INTERFACE ITest

METHOD TestMethod : BOOL
VAR_INPUT
END_VAR
END_METHOD

END_INTERFACE

(* stored: Version 1.1.0.1
   Itf ITest: Id {bfd2c572-381c-4242-a790-590066fa0848}
   Method TestMethod: Id {a7e91d8c-bcc4-4368-90b6-e02d3960ccc7} *)
